Staubli VAL3: selectItem.pgx

public program selectItem(num x_nIndex)
  local string l_sItem
begin
end
